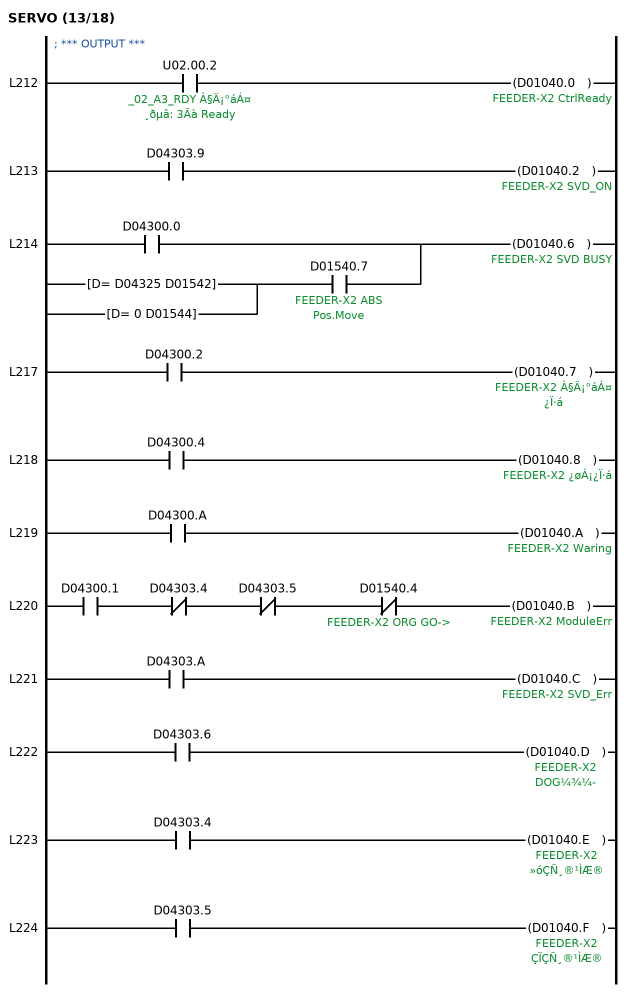
// *** OUTPUT ***
; L212
LOAD      U02.00.2	// _02_A3_RDY À§Ä¡°áÁ¤ ¸ðµâ: 3Ãà Ready
OUT       D01040.0	// FEEDER-X2 CtrlReady
; L213
LOAD      D04303.9
OUT       D01040.2	// FEEDER-X2 SVD_ON
; L214
LOAD      D04300.0
LOADD=    D04325 D01542
ORD=      0 D01544
AND       D01540.7	// FEEDER-X2 ABS Pos.Move
OR LOAD
OUT       D01040.6	// FEEDER-X2 SVD BUSY
; L217
LOAD      D04300.2
OUT       D01040.7	// FEEDER-X2 À§Ä¡°áÁ¤ ¿Ï·á
; L218
LOAD      D04300.4
OUT       D01040.8	// FEEDER-X2 ¿øÁ¡¿Ï·á
; L219
LOAD      D04300.A
OUT       D01040.A	// FEEDER-X2 Waring
; L220
LOAD      D04300.1
AND NOT   D04303.4
AND NOT   D04303.5
AND NOT   D01540.4	// FEEDER-X2 ORG GO->
OUT       D01040.B	// FEEDER-X2 ModuleErr
; L221
LOAD      D04303.A
OUT       D01040.C	// FEEDER-X2 SVD_Err
; L222
LOAD      D04303.6
OUT       D01040.D	// FEEDER-X2 DOG¼¾¼­
; L223
LOAD      D04303.4
OUT       D01040.E	// FEEDER-X2 »óÇÑ¸®¹ÌÆ®
; L224
LOAD      D04303.5
OUT       D01040.F	// FEEDER-X2 ÇÏÇÑ¸®¹ÌÆ®

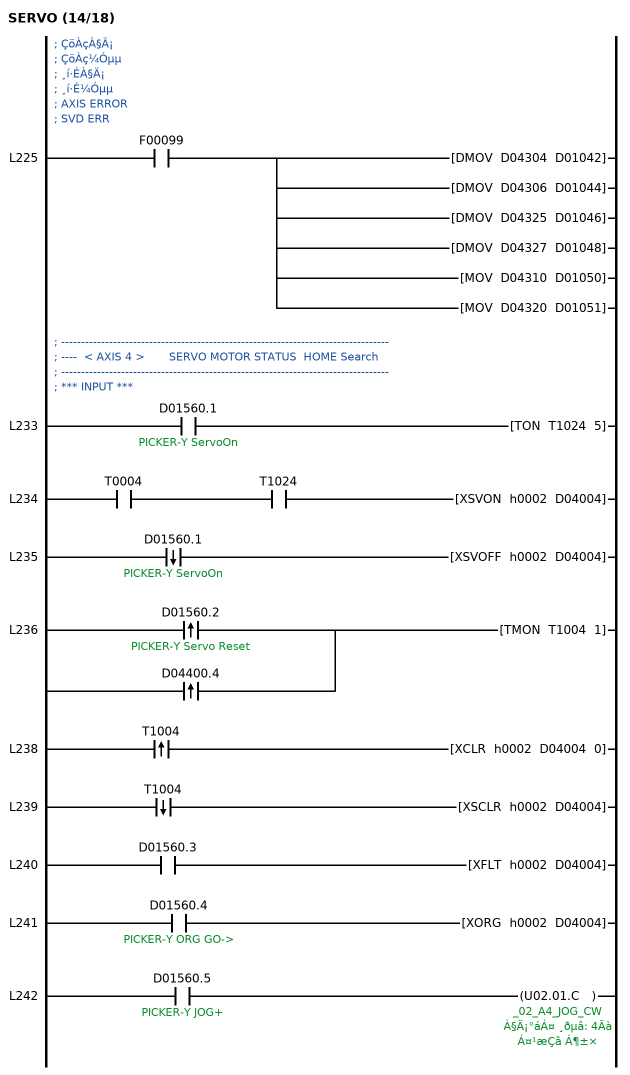
; L225
LOAD      F00099
DMOV      D04304 D01042
DMOV      D04306 D01044
DMOV      D04325 D01046
DMOV      D04327 D01048
MOV       D04310 D01050
MOV       D04320 D01051
// output comment: ÇöÀçÀ§Ä¡
// output comment: ÇöÀç¼Óµµ
// output comment: ¸í·ÉÀ§Ä¡
// output comment: ¸í·É¼Óµµ
// output comment: AXIS ERROR
// output comment: SVD ERR
// ----------------------------------------------------------------------------------
// 
// ----  < AXIS 4 >       SERVO MOTOR STATUS  HOME Search
// 
// ----------------------------------------------------------------------------------
// *** INPUT ***
; L233
LOAD      D01560.1	// PICKER-Y ServoOn
TON       T1024 5
; L234
LOAD      T0004
AND       T1024
XSVON     h0002 D04004
; L235
LOADN     D01560.1	// PICKER-Y ServoOn
XSVOFF    h0002 D04004
; L236
LOADP     D01560.2	// PICKER-Y Servo Reset
ORP       D04400.4
TMON      T1004 1
; L238
LOADP     T1004
XCLR      h0002 D04004 0
; L239
LOADN     T1004
XSCLR     h0002 D04004
; L240
LOAD      D01560.3
XFLT      h0002 D04004
; L241
LOAD      D01560.4	// PICKER-Y ORG GO->
XORG      h0002 D04004
; L242
LOAD      D01560.5	// PICKER-Y JOG+
OUT       U02.01.C	// _02_A4_JOG_CW À§Ä¡°áÁ¤ ¸ðµâ: 4Ãà Á¤¹æÇâ Á¶±×

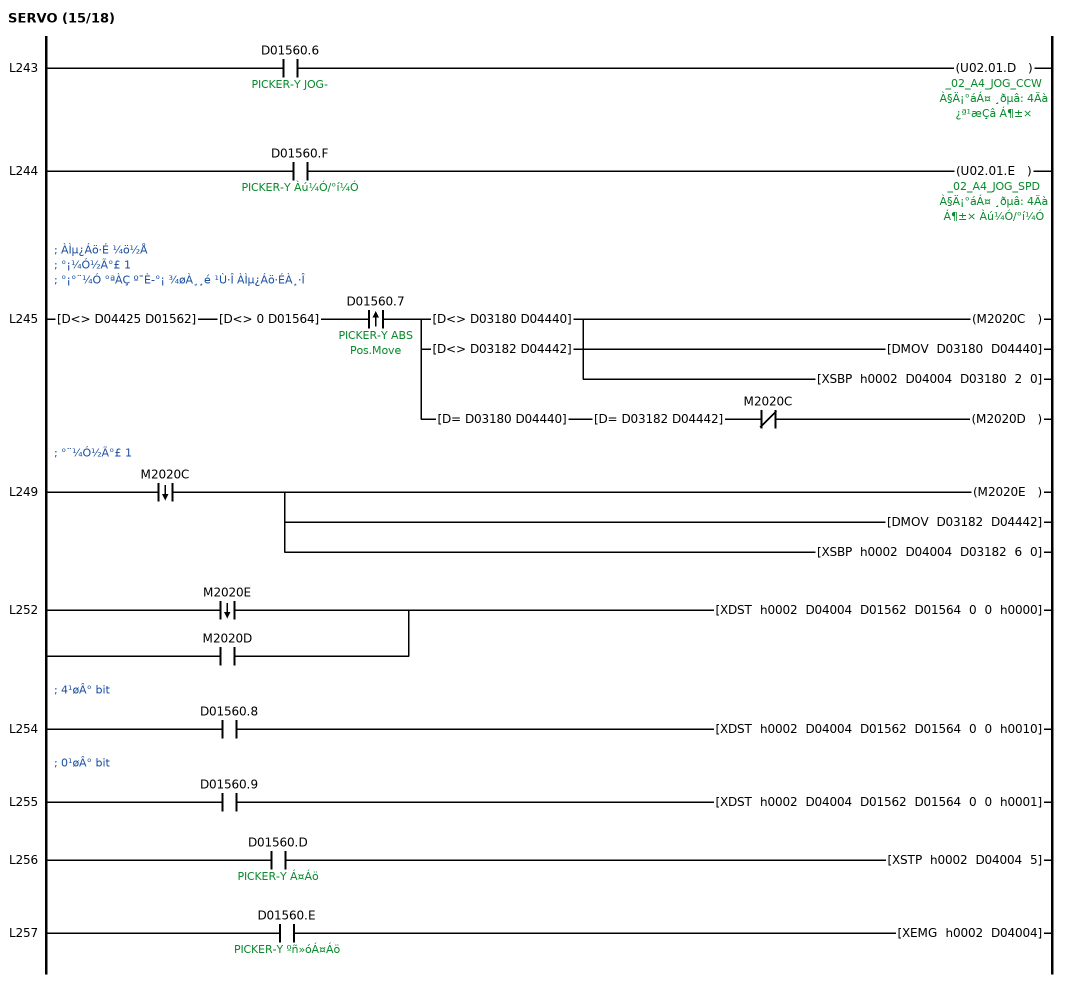
; L243
LOAD      D01560.6	// PICKER-Y JOG-
OUT       U02.01.D	// _02_A4_JOG_CCW À§Ä¡°áÁ¤ ¸ðµâ: 4Ãà ¿ª¹æÇâ Á¶±×
; L244
LOAD      D01560.F	// PICKER-Y Àú¼Ó/°í¼Ó
OUT       U02.01.E	// _02_A4_JOG_SPD À§Ä¡°áÁ¤ ¸ðµâ: 4Ãà Á¶±× Àú¼Ó/°í¼Ó
; L245
LOADD<>   D04425 D01562
ANDD<>    0 D01564
ANDP      D01560.7	// PICKER-Y ABS Pos.Move
MPUSH
LOADD<>   D03180 D04440
ORD<>     D03182 D04442
AND LOAD
OUT       M2020C
DMOV      D03180 D04440
XSBP      h0002 D04004 D03180 2 0
MPOP
ANDD=     D03180 D04440
ANDD=     D03182 D04442
AND NOT   M2020C
OUT       M2020D
// output comment: ÀÌµ¿Áö·É ¼ö½Å
// output comment: °¡¼Ó½Ã°£ 1
// output comment: °¡°¨¼Ó °ªÀÇ º¯È­°¡ ¾øÀ¸¸é ¹Ù·Î ÀÌµ¿Áö·ÉÀ¸·Î
; L249
LOADN     M2020C
OUT       M2020E
DMOV      D03182 D04442
XSBP      h0002 D04004 D03182 6 0
// output comment: °¨¼Ó½Ã°£ 1
; L252
LOADN     M2020E
OR        M2020D
XDST      h0002 D04004 D01562 D01564 0 0 h0000
; L254
LOAD      D01560.8
XDST      h0002 D04004 D01562 D01564 0 0 h0010
// output comment: 4¹øÂ° bit
; L255
LOAD      D01560.9
XDST      h0002 D04004 D01562 D01564 0 0 h0001
// output comment: 0¹øÂ° bit
; L256
LOAD      D01560.D	// PICKER-Y Á¤Áö
XSTP      h0002 D04004 5
; L257
LOAD      D01560.E	// PICKER-Y ºñ»óÁ¤Áö
XEMG      h0002 D04004

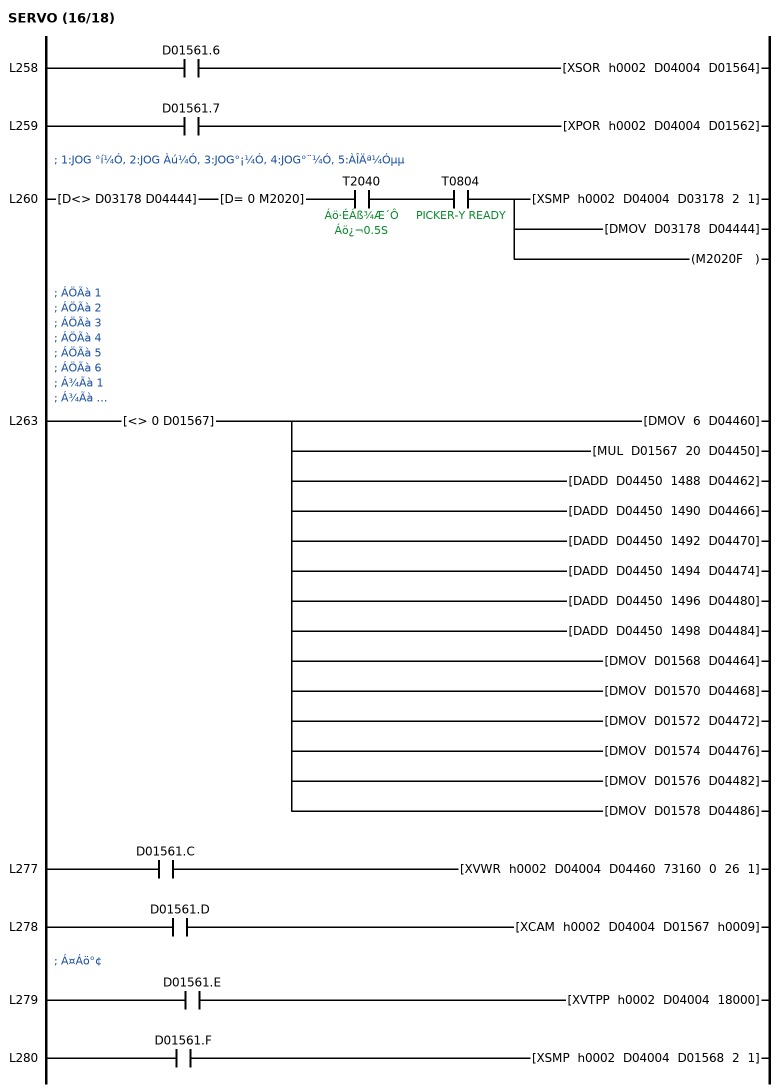
; L258
LOAD      D01561.6
XSOR      h0002 D04004 D01564
; L259
LOAD      D01561.7
XPOR      h0002 D04004 D01562
; L260
LOADD<>   D03178 D04444
ANDD=     0 M2020
AND       T2040	// Áö·ÉÁß¾Æ´Ô Áö¿¬0.5S
AND       T0804	// PICKER-Y READY
XSMP      h0002 D04004 D03178 2 1
DMOV      D03178 D04444
OUT       M2020F
// output comment: 1:JOG °í¼Ó, 2:JOG Àú¼Ó, 3:JOG°¡¼Ó, 4:JOG°¨¼Ó, 5:ÀÎÄª¼Óµµ
; L263
LOAD<>    0 D01567
DMOV      6 D04460
MUL       D01567 20 D04450
DADD      D04450 1488 D04462
DADD      D04450 1490 D04466
DADD      D04450 1492 D04470
DADD      D04450 1494 D04474
DADD      D04450 1496 D04480
DADD      D04450 1498 D04484
DMOV      D01568 D04464
DMOV      D01570 D04468
DMOV      D01572 D04472
DMOV      D01574 D04476
DMOV      D01576 D04482
DMOV      D01578 D04486
// output comment: ÁÖÃà 1
// output comment: ÁÖÃà 2
// output comment: ÁÖÃà 3
// output comment: ÁÖÃà 4
// output comment: ÁÖÃà 5
// output comment: ÁÖÃà 6
// output comment: Á¾Ãà 1
// output comment: Á¾Ãà 2
// output comment: Á¾Ãà 3
// output comment: Á¾Ãà 4
// output comment: Á¾Ãà 5
// output comment: Á¾Ãà 6
; L277
LOAD      D01561.C
XVWR      h0002 D04004 D04460 73160 0 26 1
; L278
LOAD      D01561.D
XCAM      h0002 D04004 D01567 h0009
; L279
LOAD      D01561.E
XVTPP     h0002 D04004 18000
// output comment: Á¤Áö°¢
; L280
LOAD      D01561.F
XSMP      h0002 D04004 D01568 2 1

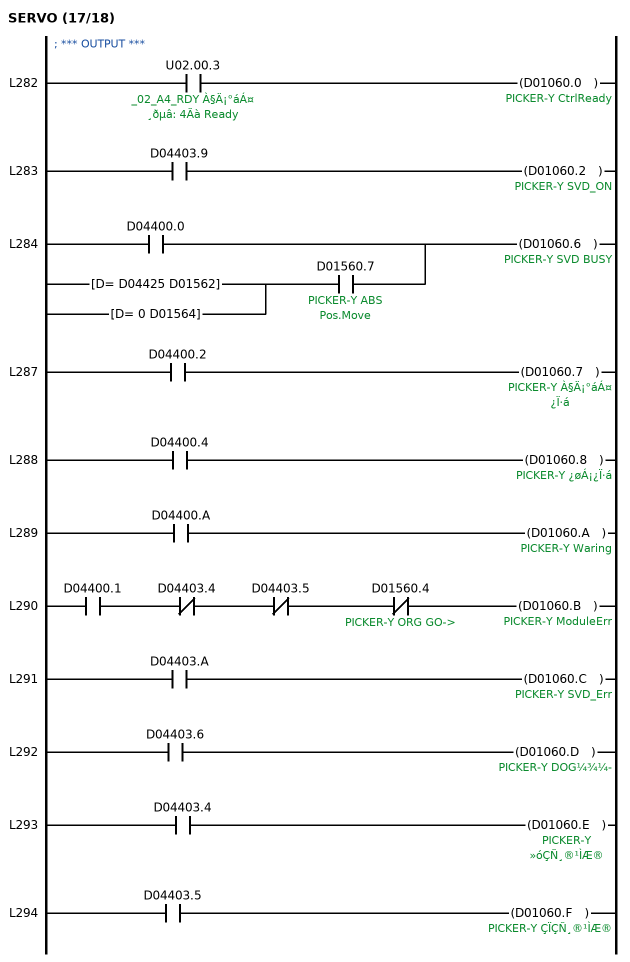
// *** OUTPUT ***
; L282
LOAD      U02.00.3	// _02_A4_RDY À§Ä¡°áÁ¤ ¸ðµâ: 4Ãà Ready
OUT       D01060.0	// PICKER-Y CtrlReady
; L283
LOAD      D04403.9
OUT       D01060.2	// PICKER-Y SVD_ON
; L284
LOAD      D04400.0
LOADD=    D04425 D01562
ORD=      0 D01564
AND       D01560.7	// PICKER-Y ABS Pos.Move
OR LOAD
OUT       D01060.6	// PICKER-Y SVD BUSY
; L287
LOAD      D04400.2
OUT       D01060.7	// PICKER-Y À§Ä¡°áÁ¤ ¿Ï·á
; L288
LOAD      D04400.4
OUT       D01060.8	// PICKER-Y ¿øÁ¡¿Ï·á
; L289
LOAD      D04400.A
OUT       D01060.A	// PICKER-Y Waring
; L290
LOAD      D04400.1
AND NOT   D04403.4
AND NOT   D04403.5
AND NOT   D01560.4	// PICKER-Y ORG GO->
OUT       D01060.B	// PICKER-Y ModuleErr
; L291
LOAD      D04403.A
OUT       D01060.C	// PICKER-Y SVD_Err
; L292
LOAD      D04403.6
OUT       D01060.D	// PICKER-Y DOG¼¾¼­
; L293
LOAD      D04403.4
OUT       D01060.E	// PICKER-Y »óÇÑ¸®¹ÌÆ®
; L294
LOAD      D04403.5
OUT       D01060.F	// PICKER-Y ÇÏÇÑ¸®¹ÌÆ®

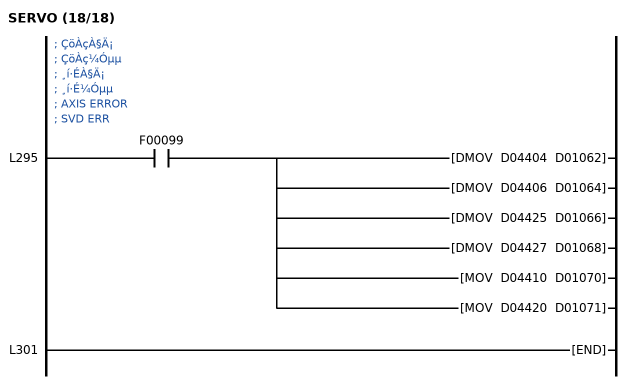
; L295
LOAD      F00099
DMOV      D04404 D01062
DMOV      D04406 D01064
DMOV      D04425 D01066
DMOV      D04427 D01068
MOV       D04410 D01070
MOV       D04420 D01071
// output comment: ÇöÀçÀ§Ä¡
// output comment: ÇöÀç¼Óµµ
// output comment: ¸í·ÉÀ§Ä¡
// output comment: ¸í·É¼Óµµ
// output comment: AXIS ERROR
// output comment: SVD ERR
; L301
END

PROGRAM INTERFACE (task: ½ºÄµ ÇÁ·Î±×·¥)

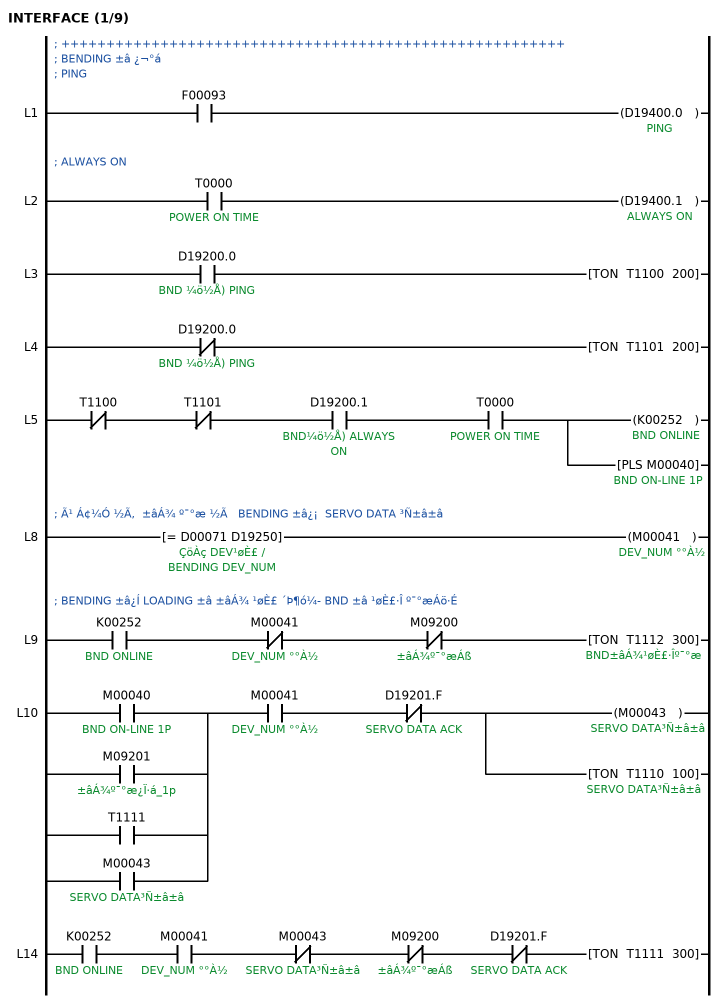
// ++++++++++++++++++++++++++++++++++++++++++++++++++++++++
//    BENDING ±â ¿¬°á
; L1
LOAD      F00093
OUT       D19400.0	// PING
// output comment: PING
; L2
LOAD      T0000	// POWER ON TIME
OUT       D19400.1	// ALWAYS ON
// output comment: ALWAYS ON
; L3
LOAD      D19200.0	// BND ¼ö½Å) PING
TON       T1100 200
; L4
LOAD NOT  D19200.0	// BND ¼ö½Å) PING
TON       T1101 200
; L5
LOAD NOT  T1100
AND NOT   T1101
AND       D19200.1	// BND¼ö½Å) ALWAYS ON
AND       T0000	// POWER ON TIME
OUT       K00252	// BND ONLINE
OUTP      M00040	// BND ON-LINE 1P
// Ã¹ Á¢¼Ó ½Ã,  ±âÁ¾ º¯°æ ½Ã   BENDING ±â¿¡  SERVO DATA ³Ñ±â±â
; L8
LOAD=     D00071 D19250	// ÇöÀç DEV¹øÈ£ / BENDING DEV_NUM
OUT       M00041	// DEV_NUM °°À½
; L9
LOAD      K00252	// BND ONLINE
AND NOT   M00041	// DEV_NUM °°À½
AND NOT   M09200	// ±âÁ¾º¯°æÁß
TON       T1112 300	// BND±âÁ¾¹øÈ£·Îº¯°æ
// output comment: BENDING ±â¿Í LOADING ±â ±âÁ¾ ¹øÈ£ ´Þ¶ó¼­ BND ±â ¹øÈ£·Î º¯°æÁö·É
; L10
LOAD      M00040	// BND ON-LINE 1P
OR        M09201	// ±âÁ¾º¯°æ¿Ï·á_1p
OR        T1111
OR        M00043	// SERVO DATA³Ñ±â±â
AND       M00041	// DEV_NUM °°À½
AND NOT   D19201.F	// SERVO DATA ACK
OUT       M00043	// SERVO DATA³Ñ±â±â
TON       T1110 100	// SERVO DATA³Ñ±â±â
; L14
LOAD      K00252	// BND ONLINE
AND       M00041	// DEV_NUM °°À½
AND NOT   M00043	// SERVO DATA³Ñ±â±â
AND NOT   M09200	// ±âÁ¾º¯°æÁß
AND NOT   D19201.F	// SERVO DATA ACK
TON       T1111 300

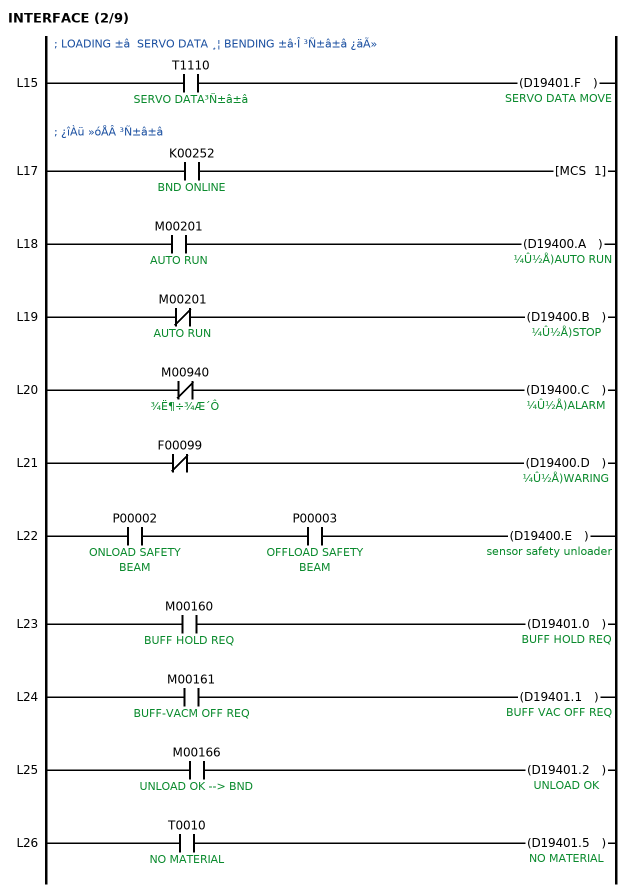
; L15
LOAD      T1110	// SERVO DATA³Ñ±â±â
OUT       D19401.F	// SERVO DATA MOVE
// output comment: LOADING ±â  SERVO DATA ¸¦ BENDING ±â·Î ³Ñ±â±â ¿äÃ»
// ¿îÀü »óÅÂ ³Ñ±â±â
; L17
LOAD      K00252	// BND ONLINE
MCS       1
; L18
LOAD      M00201	// AUTO RUN
OUT       D19400.A	// ¼Û½Å)AUTO RUN
; L19
LOAD NOT  M00201	// AUTO RUN
OUT       D19400.B	// ¼Û½Å)STOP
; L20
LOAD NOT  M00940	// ¾Ë¶÷¾Æ´Ô
OUT       D19400.C	// ¼Û½Å)ALARM
; L21
LOAD NOT  F00099
OUT       D19400.D	// ¼Û½Å)WARING
; L22
LOAD      P00002	// ONLOAD SAFETY BEAM
AND       P00003	// OFFLOAD SAFETY BEAM
OUT       D19400.E	// sensor safety unloader
; L23
LOAD      M00160	// BUFF HOLD REQ
OUT       D19401.0	// BUFF HOLD REQ
; L24
LOAD      M00161	// BUFF-VACM OFF REQ
OUT       D19401.1	// BUFF VAC OFF REQ
; L25
LOAD      M00166	// UNLOAD OK --> BND
OUT       D19401.2	// UNLOAD OK
; L26
LOAD      T0010	// NO MATERIAL
OUT       D19401.5	// NO MATERIAL

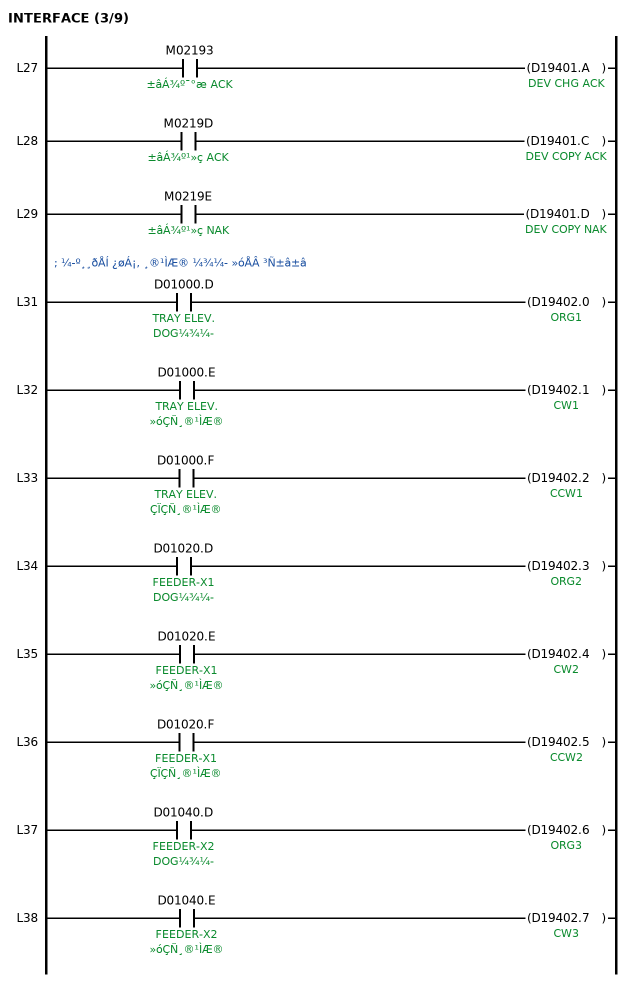
; L27
LOAD      M02193	// ±âÁ¾º¯°æ ACK
OUT       D19401.A	// DEV CHG ACK
; L28
LOAD      M0219D	// ±âÁ¾º¹»ç ACK
OUT       D19401.C	// DEV COPY ACK
; L29
LOAD      M0219E	// ±âÁ¾º¹»ç NAK
OUT       D19401.D	// DEV COPY NAK
// ¼­º¸¸ðÅÍ ¿øÁ¡, ¸®¹ÌÆ® ¼¾¼­ »óÅÂ ³Ñ±â±â
; L31
LOAD      D01000.D	// TRAY ELEV. DOG¼¾¼­
OUT       D19402.0	// ORG1
; L32
LOAD      D01000.E	// TRAY ELEV. »óÇÑ¸®¹ÌÆ®
OUT       D19402.1	// CW1
; L33
LOAD      D01000.F	// TRAY ELEV. ÇÏÇÑ¸®¹ÌÆ®
OUT       D19402.2	// CCW1
; L34
LOAD      D01020.D	// FEEDER-X1 DOG¼¾¼­
OUT       D19402.3	// ORG2
; L35
LOAD      D01020.E	// FEEDER-X1 »óÇÑ¸®¹ÌÆ®
OUT       D19402.4	// CW2
; L36
LOAD      D01020.F	// FEEDER-X1 ÇÏÇÑ¸®¹ÌÆ®
OUT       D19402.5	// CCW2
; L37
LOAD      D01040.D	// FEEDER-X2 DOG¼¾¼­
OUT       D19402.6	// ORG3
; L38
LOAD      D01040.E	// FEEDER-X2 »óÇÑ¸®¹ÌÆ®
OUT       D19402.7	// CW3

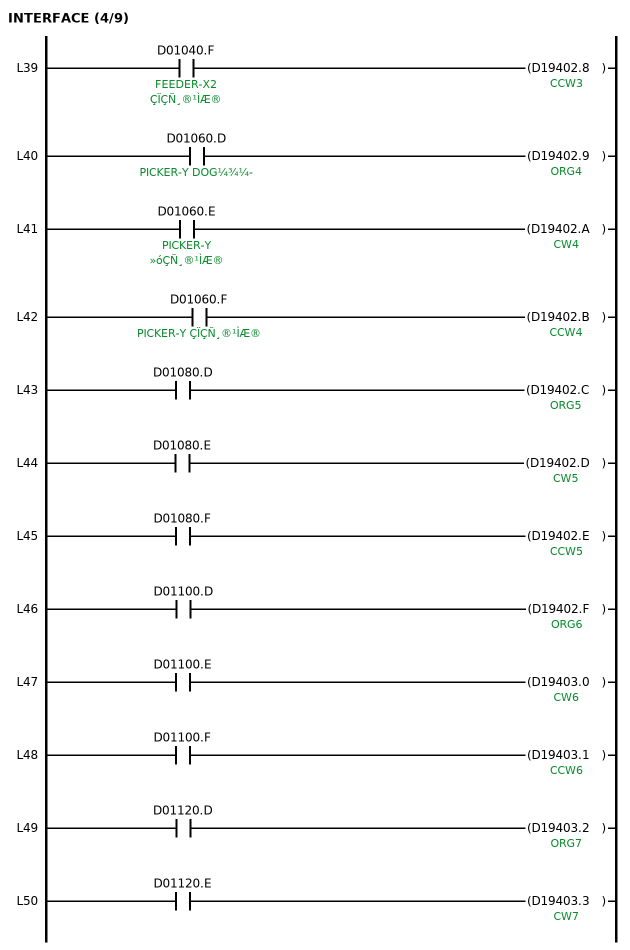
; L39
LOAD      D01040.F	// FEEDER-X2 ÇÏÇÑ¸®¹ÌÆ®
OUT       D19402.8	// CCW3
; L40
LOAD      D01060.D	// PICKER-Y DOG¼¾¼­
OUT       D19402.9	// ORG4
; L41
LOAD      D01060.E	// PICKER-Y »óÇÑ¸®¹ÌÆ®
OUT       D19402.A	// CW4
; L42
LOAD      D01060.F	// PICKER-Y ÇÏÇÑ¸®¹ÌÆ®
OUT       D19402.B	// CCW4
; L43
LOAD      D01080.D
OUT       D19402.C	// ORG5
; L44
LOAD      D01080.E
OUT       D19402.D	// CW5
; L45
LOAD      D01080.F
OUT       D19402.E	// CCW5
; L46
LOAD      D01100.D
OUT       D19402.F	// ORG6
; L47
LOAD      D01100.E
OUT       D19403.0	// CW6
; L48
LOAD      D01100.F
OUT       D19403.1	// CCW6
; L49
LOAD      D01120.D
OUT       D19403.2	// ORG7
; L50
LOAD      D01120.E
OUT       D19403.3	// CW7

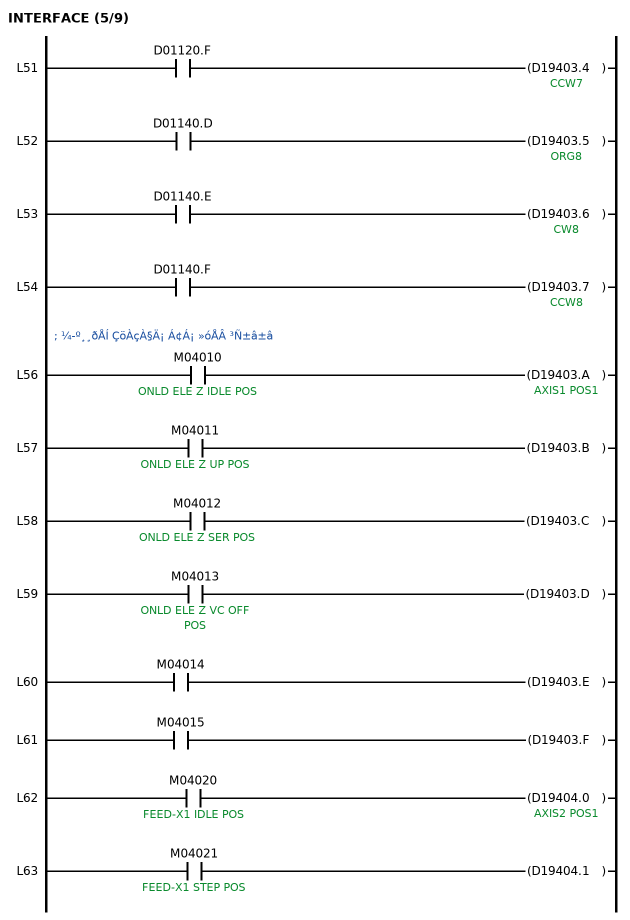
; L51
LOAD      D01120.F
OUT       D19403.4	// CCW7
; L52
LOAD      D01140.D
OUT       D19403.5	// ORG8
; L53
LOAD      D01140.E
OUT       D19403.6	// CW8
; L54
LOAD      D01140.F
OUT       D19403.7	// CCW8
// ¼­º¸¸ðÅÍ ÇöÀçÀ§Ä¡ Á¢Á¡ »óÅÂ ³Ñ±â±â
; L56
LOAD      M04010	// ONLD ELE Z IDLE POS
OUT       D19403.A	// AXIS1 POS1
; L57
LOAD      M04011	// ONLD ELE Z UP POS
OUT       D19403.B
; L58
LOAD      M04012	// ONLD ELE Z SER POS
OUT       D19403.C
; L59
LOAD      M04013	// ONLD ELE Z VC OFF POS
OUT       D19403.D
; L60
LOAD      M04014
OUT       D19403.E
; L61
LOAD      M04015
OUT       D19403.F
; L62
LOAD      M04020	// FEED-X1 IDLE POS
OUT       D19404.0	// AXIS2 POS1
; L63
LOAD      M04021	// FEED-X1 STEP POS
OUT       D19404.1

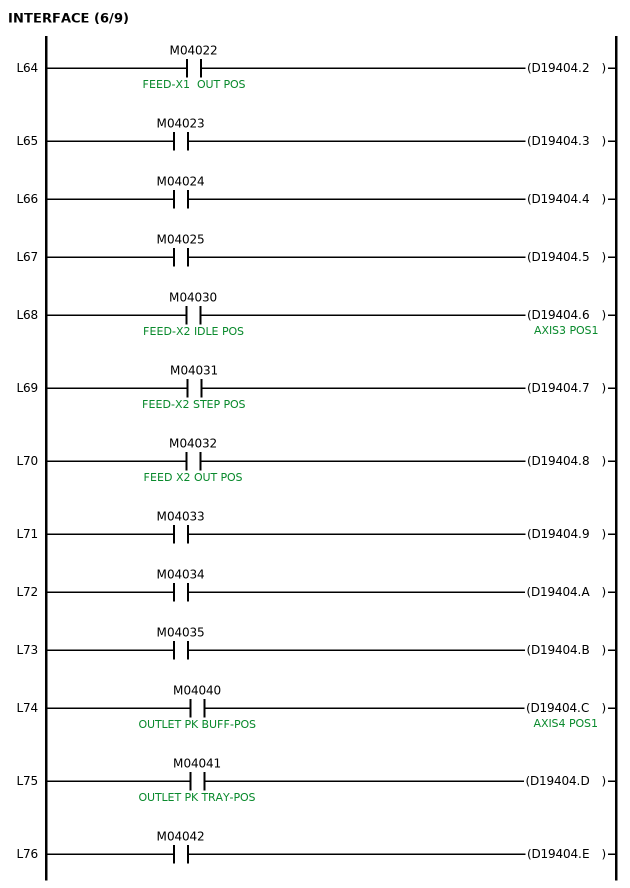
; L64
LOAD      M04022	// FEED-X1  OUT POS
OUT       D19404.2
; L65
LOAD      M04023
OUT       D19404.3
; L66
LOAD      M04024
OUT       D19404.4
; L67
LOAD      M04025
OUT       D19404.5
; L68
LOAD      M04030	// FEED-X2 IDLE POS
OUT       D19404.6	// AXIS3 POS1
; L69
LOAD      M04031	// FEED-X2 STEP POS
OUT       D19404.7
; L70
LOAD      M04032	// FEED X2 OUT POS
OUT       D19404.8
; L71
LOAD      M04033
OUT       D19404.9
; L72
LOAD      M04034
OUT       D19404.A
; L73
LOAD      M04035
OUT       D19404.B
; L74
LOAD      M04040	// OUTLET PK BUFF-POS
OUT       D19404.C	// AXIS4 POS1
; L75
LOAD      M04041	// OUTLET PK TRAY-POS
OUT       D19404.D
; L76
LOAD      M04042
OUT       D19404.E

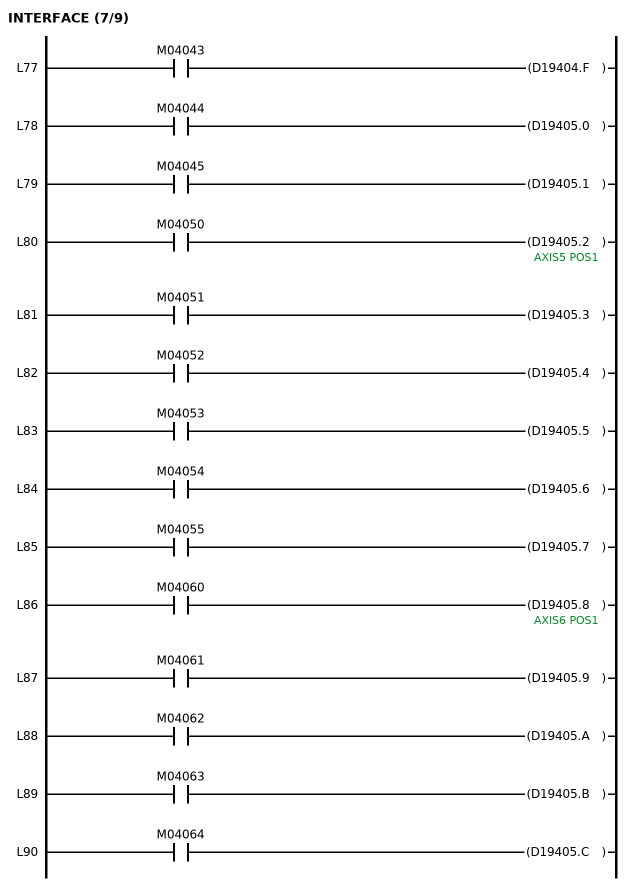
; L77
LOAD      M04043
OUT       D19404.F
; L78
LOAD      M04044
OUT       D19405.0
; L79
LOAD      M04045
OUT       D19405.1
; L80
LOAD      M04050
OUT       D19405.2	// AXIS5 POS1
; L81
LOAD      M04051
OUT       D19405.3
; L82
LOAD      M04052
OUT       D19405.4
; L83
LOAD      M04053
OUT       D19405.5
; L84
LOAD      M04054
OUT       D19405.6
; L85
LOAD      M04055
OUT       D19405.7
; L86
LOAD      M04060
OUT       D19405.8	// AXIS6 POS1
; L87
LOAD      M04061
OUT       D19405.9
; L88
LOAD      M04062
OUT       D19405.A
; L89
LOAD      M04063
OUT       D19405.B
; L90
LOAD      M04064
OUT       D19405.C

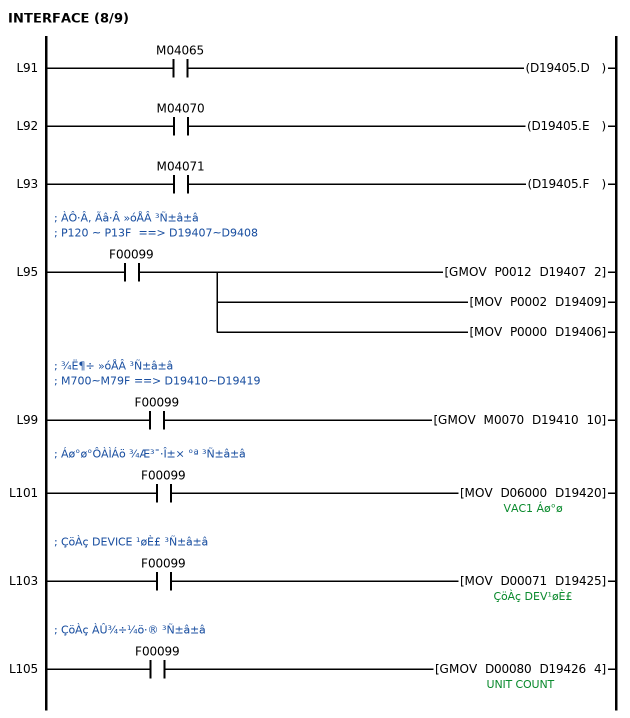
; L91
LOAD      M04065
OUT       D19405.D
; L92
LOAD      M04070
OUT       D19405.E
; L93
LOAD      M04071
OUT       D19405.F
// ÀÔ·Â, Ãâ·Â »óÅÂ ³Ñ±â±â
; L95
LOAD      F00099
GMOV      P0012 D19407 2
MOV       P0002 D19409
MOV       P0000 D19406
// output comment: P120 ~ P13F  ==> D19407~D9408
// ¾Ë¶÷ »óÅÂ ³Ñ±â±â
; L99
LOAD      F00099
GMOV      M0070 D19410 10
// output comment: M700~M79F ==> D19410~D19419
// Áø°ø°ÔÀÌÁö ¾Æ³¯·Î±× °ª ³Ñ±â±â
; L101
LOAD      F00099
MOV       D06000 D19420	// VAC1 Áø°ø
// ÇöÀç DEVICE ¹øÈ£ ³Ñ±â±â
; L103
LOAD      F00099
MOV       D00071 D19425	// ÇöÀç DEV¹øÈ£
// ÇöÀç ÀÛ¾÷¼ö·® ³Ñ±â±â
; L105
LOAD      F00099
GMOV      D00080 D19426 4	// UNIT COUNT

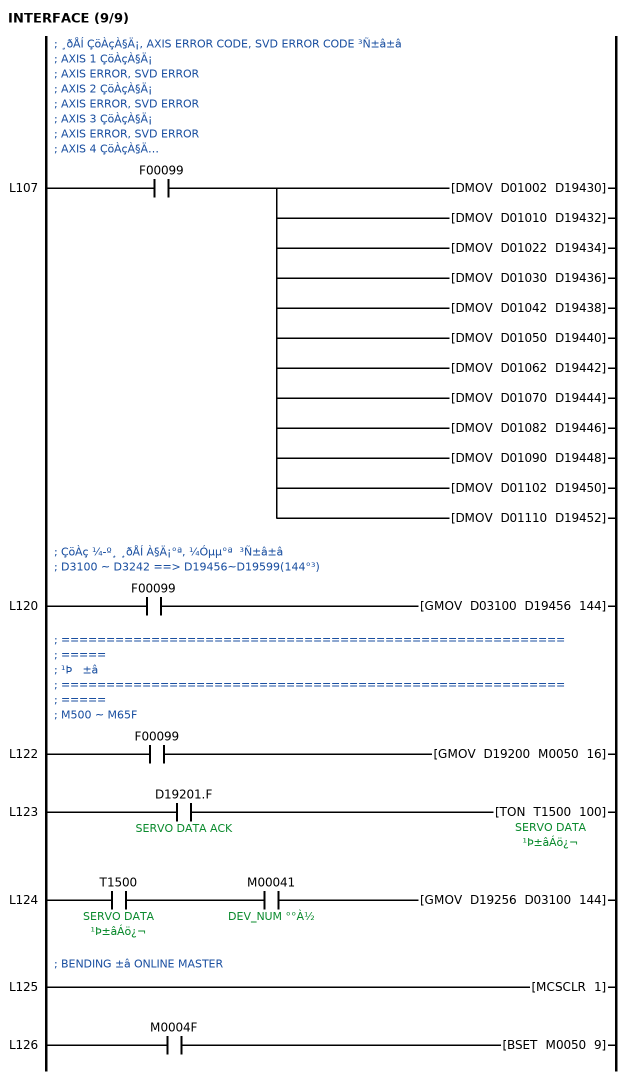
// ¸ðÅÍ ÇöÀçÀ§Ä¡, AXIS ERROR CODE, SVD ERROR CODE ³Ñ±â±â
; L107
LOAD      F00099
DMOV      D01002 D19430
DMOV      D01010 D19432
DMOV      D01022 D19434
DMOV      D01030 D19436
DMOV      D01042 D19438
DMOV      D01050 D19440
DMOV      D01062 D19442
DMOV      D01070 D19444
DMOV      D01082 D19446
DMOV      D01090 D19448
DMOV      D01102 D19450
DMOV      D01110 D19452
// output comment: AXIS 1 ÇöÀçÀ§Ä¡
// output comment: AXIS ERROR, SVD ERROR
// output comment: AXIS 2 ÇöÀçÀ§Ä¡
// output comment: AXIS ERROR, SVD ERROR
// output comment: AXIS 3 ÇöÀçÀ§Ä¡
// output comment: AXIS ERROR, SVD ERROR
// output comment: AXIS 4 ÇöÀçÀ§Ä¡
// output comment: AXIS ERROR, SVD ERROR
// output comment: AXIS 5 ÇöÀçÀ§Ä¡
// output comment: AXIS ERROR, SVD ERROR
// output comment: AXIS 6 ÇöÀçÀ§Ä¡
// output comment: AXIS ERROR, SVD ERROR
// ÇöÀç ¼­º¸ ¸ðÅÍ À§Ä¡°ª, ¼Óµµ°ª  ³Ñ±â±â
; L120
LOAD      F00099
GMOV      D03100 D19456 144
// output comment: D3100 ~ D3242 ==> D19456~D19599(144°³)
// =============================================================
// 
// 
//       ¹Þ   ±â
//       
//       
// =============================================================
; L122
LOAD      F00099
GMOV      D19200 M0050 16
// output comment: M500 ~ M65F
; L123
LOAD      D19201.F	// SERVO DATA ACK
TON       T1500 100	// SERVO DATA ¹Þ±âÁö¿¬
; L124
LOAD      T1500	// SERVO DATA ¹Þ±âÁö¿¬
AND       M00041	// DEV_NUM °°À½
GMOV      D19256 D03100 144
; L125
MCSCLR    1
// output comment: BENDING ±â ONLINE MASTER
; L126
LOAD      M0004F
BSET      M0050 9

VARIABLES AND COMMENTS (devices not used above)
D01000.1	BIT	TRAY ELEV. SVDÁØºñ»óÅÂ
D01000.4	BIT	TRAY ELEV. reset Áö·É¿Ï·á
D01000.9	BIT	TRAY ELEV. StopCommd
D01020.1	BIT	FEEDER-X1 SVDÁØºñ»óÅÂ
D01020.4	BIT	FEEDER-X1 reset Áö·É¿Ï·á
D01020.9	BIT	FEEDER-X1 StopCommd
D01040.1	BIT	FEEDER-X2 SVDÁØºñ»óÅÂ
D01040.4	BIT	FEEDER-X2 reset Áö·É¿Ï·á
D01040.9	BIT	FEEDER-X2 StopCommd
D01060.1	BIT	PICKER-Y SVDÁØºñ»óÅÂ
D01060.4	BIT	PICKER-Y reset Áö·É¿Ï·á
D01060.9	BIT	PICKER-Y StopCommd
P00137	BIT	ONLOAD TRAY SIDE CLAMP CLOSE
M00560	BIT	¼Ó¼Ò¼ÂÆÃ¿ë °­Á¦Ãâ·Â1
M00726	BIT	-
M0078A	BIT	INLET 4th PICKER VACUUM 4 ALARM
M0078B	BIT	INLET 5th PICKER VACUUM 5 ALARM